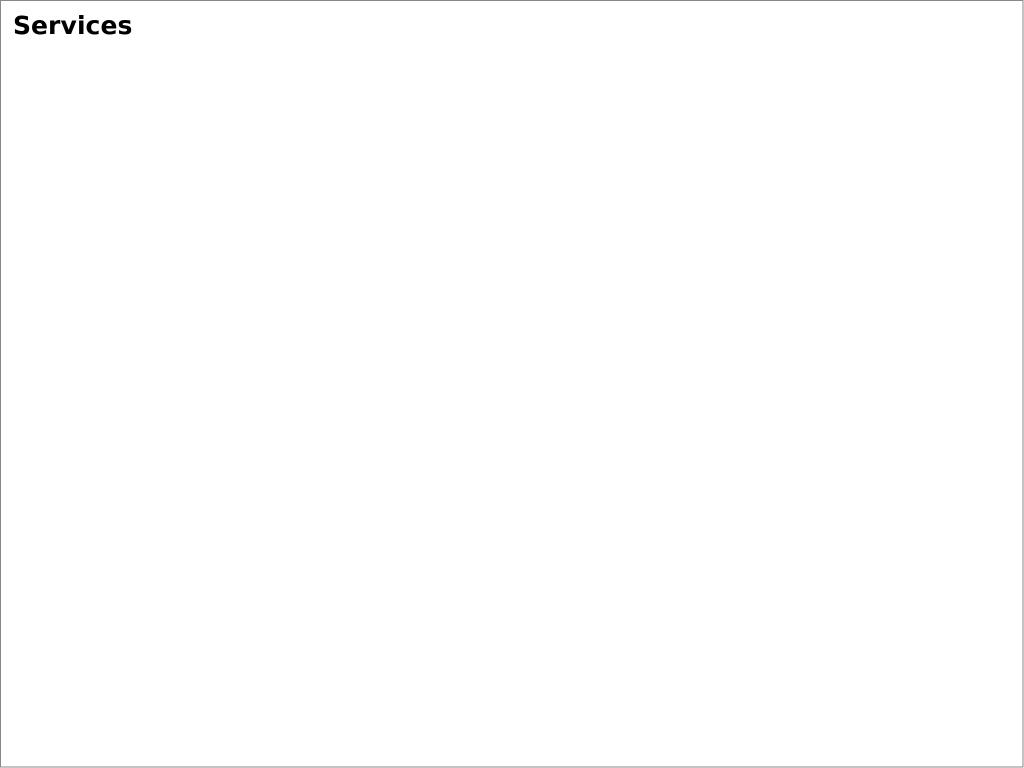
VISUALIZATION VISU_HMI_SERVICES  // 1024x768
VAR_IN_OUT
	m_Instance : FB_SERVICES;
    //m_Hmi : FB_HMI_SERVICES;
END_VAR
    Label (10,10 150x30), "Services"
END_VISUALIZATION

(* stored: Version 1.1.0.1, ProductVersion 3.1.4024.14
   Visu VISU_HMI_SERVICES: Id {5161b964-0023-49c1-b85d-6675b7e31a31} *)
